PROGRAM MAIN
VAR
	PBSTart: BOOL;
	PBStop: BOOL;
	Motor: BOOL;
END_VAR

IF PBSTop THEN
	Motor:= FALSE;
ELSIF PBSTart THEN
	Motor:= TRUE;
END_IF

END_PROGRAM

(* stored: Version 1.1.0.1, ProductVersion 3.1.4024.12
   POU MAIN: Id {a2d77e32-9531-4294-a721-76b547fe715a}, SpecialFunc None *)
